# EPICS substitutions: dg535/dg535App/Db/userHost.substitutions
# Example substitutions file

file "db/dbExample1.db" {
    { user = "roryHost" }
}

file db/dbExample2.db {
    pattern { user, no, scan }
        { "roryHost", 1, "1 second" }
        { "roryHost", 2, "2 second" }
        { "roryHost", 3, "5 second" }
}
